Staubli VAL3: getToolStatus.pgx

program getToolStatus(string& x_sStatus (dimensions=1))
begin
  // This program returns the status of the tool
  //
  // Input parameters
  //  None            :
  //
  // Output parameters
  //  x_sStatus       : Status of the tool
  //     "Part_taken" = There is a part on the tool
  //         "Vacuum" = Vacuum is on
  //           "Blow" = Blow is on
  //            "Off" = The tool is not activated
  //
  //----------------------------------------------------------------
  //
  if dBlow==false and dVacuum==true and dPartInTool==true
    x_sStatus="PartInTool"
  elseIf dBlow==false and dVacuum==true
    x_sStatus="Vacuum"
  elseIf dBlow==true
    x_sStatus="Blow"
  elseIf dBlow==false and dVacuum==false
    x_sStatus="Off"
  else
    //default reset to off
    x_sStatus="off"
    dVacuum=false
    dBlow=false
  endIf
end
